RoboDK station: KUKA.rdk

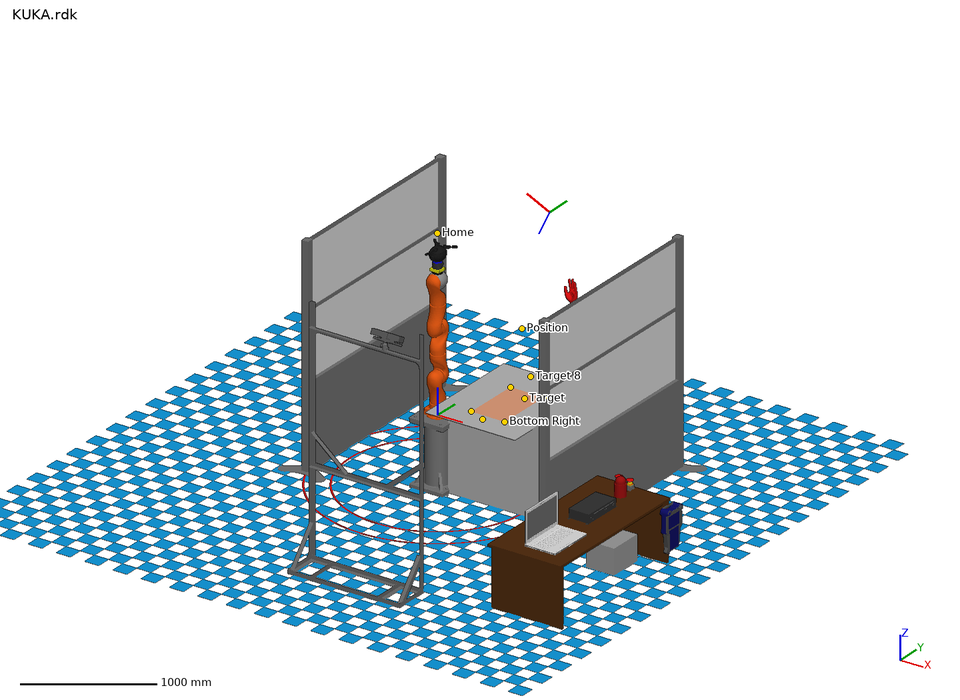
[picture v0: the station drawn from its stored meshes, robots at their saved joint values, targets as dots, program paths as lines]
Station robotSim. Poses are relative to the parent item; angles as X-Y-Z fixed-axis rotations.
Station parameters (name, value as stored): IO_5, 1
  - frame KUKA-LWR-IV-PLUS Base at (0, 0, 570) mm
    - robot KUKA: 7 axes
        modified DH rows (alpha deg, a mm, theta deg, d mm): 0, 0, 0, 310.5; -90, 0, -90, 0; 90, 0, 0, 400; -90, 0, 0, 0; 90, 0, 0, 390; -90, 0, 0, 0; 90, 0, 0, 78
        joint limits [-170, -30, -170, -120, -170, -120, -170] to [170, 210, 170, 120, 170, 120, 170]; home [0, 90, 0, 0, 0, 0, 0]; saved at [0, 90, 0, 0, 0, 0, 0]
      - tool Gripper, TCP at (0, 0, 300) mm, size 214.4 x 261.8 x 207.2 mm, geometry from FULL_GRIPPER_ATI.stl
    - target Target (Cartesian target) at (600, 250, 200) mm, rotated rx -90 ry 0 rz 0 deg; joints [-12.043, 152.871, 0, -75.808, -99.102, -97.918, -49.31] of KUKA
    - target Bottom Right (Cartesian target) at (705, -150, 200) mm, rotated rx 180 ry 0 rz -135 deg; joints [-12.011, 146.511, 0, -26.598, 0, 96.891, -57.011] of KUKA
    - target Bottom Left (Cartesian target) at (405, -150, 200) mm, rotated rx 180 ry 0 rz 135 deg; joints [-20.323, 99.106, 0, -99.97, 0, 70.924, 24.677] of KUKA
    - target Top Left (Cartesian target) at (405, 350, 200) mm, rotated rx 180 ry 0 rz 45 deg; joints [-139.167, 66.69, 0, 81.525, 0, -75.165, -4.167] of KUKA
    - target Top Right (Cartesian target) at (705, 350, 200) mm, rotated rx 180 ry 0 rz -45 deg; joints [-134.648, 29.334, 0, 17.033, 0, -102.301, 90.352] of KUKA
    - target Position (Cartesian target) at (570, 260, 760) mm, rotated rx -90 ry 0 rz 0 deg; joints [-7.407, 162.566, 0, 37.615, 96.082, 94.235, -124.726] of KUKA
    - target Target 8 (Cartesian target) at (585, 350, 335) mm, rotated rx 180 ry 0 rz 45 deg; joints [-150.368, 51.861, 0, 38.836, 0, -103.025, -15.368] of KUKA
    - frame Light Source at (1000, 0, 1930) mm, rotated rx 180 ry -25 rz 180 deg
    - target Test (joint target) at (545, -205, 200) mm, rotated rx 165 ry 0 rz 45 deg; joints [-15.931, 108.28, 0, -90.444, -8.492, 58.378, 122.709] of KUKA
    - target Home (Cartesian target) at (0, 0, 1478.5) mm; joints [0, 90, 0, 0, 0, 0, 0] of KUKA
    - object Sheet at (555, 100, 200) mm, rotated rx 0 ry 0 rz 90 deg, size 500 x 300 x 0.1 mm, geometry from Sheet.stl
  - object Base at (0, 0, 0) mm, size 305 x 305 x 604 mm, geometry from Base.stl
  - object Plane at (0, 0, 0) mm, size 5042.2 x 5042.2 x 2.5 mm, geometry from plane_1m_grid.sld
  - object ATI_FT_Controller at (1800, -600, 520) mm, rotated rx 0 ry 0 rz -90 deg, size 383.6 x 183 x 76 mm, geometry from ATI_FT_Controller.stl
  - object Kinect at (620, -1500, 1985) mm, rotated rx -119.64 ry 0 rz 0 deg, size 250 x 70 x 76 mm, geometry from Kinect.stl
  - object Camera_Base at (620, -1560, 1962) mm, rotated rx 0 ry 0 rz -90 deg, size 300 x 1000 x 2100 mm, geometry from Camera_Base.stl
  - object Wall1 at (1270, 400, 0) mm, rotated rx 0 ry 0 rz 90 deg, size 1940 x 400 x 1880 mm, geometry from Wall_stripped.stl
  - object Glass1.1 at (1270, 400, 1008) mm, rotated rx 0 ry 0 rz 90 deg, size 1640 x 10 x 555 mm, geometry from Glass1.stl
  - object Glass1.2 at (1270, 400, 1582) mm, rotated rx 0 ry 0 rz 90 deg, size 1640 x 10 x 535 mm, geometry from Glass2.stl
  - object Wall2 at (-920, 500, 0) mm, rotated rx 0 ry 0 rz 90 deg, size 1940 x 400 x 1880 mm, geometry from Wall_stripped.stl
  - object Glass2.1 at (-920, 500, 1008) mm, rotated rx 0 ry 0 rz 90 deg, size 1640 x 10 x 555 mm, geometry from Glass1.stl
  - object Glass2.2 at (-920, 500, 1582) mm, rotated rx 0 ry 0 rz 90 deg, size 1640 x 10 x 535 mm, geometry from Glass2.stl
  - object Table at (535, 150, 0) mm, size 800 x 1000 x 770 mm, geometry from Table.stl
  - object Desk at (1800, -770, 520) mm, rotated rx 0 ry 0 rz -90 deg, size 1400 x 650 x 520 mm, geometry from Desk.stl
  - object Laptop at (2000, -950, 520) mm, rotated rx 90 ry 0 rz 90 deg, size 411 x 298 x 272.1 mm, geometry from Laptop.stl
  - object Safety Light at (1800, -250, 470) mm, rotated rx 90 ry 0 rz 0 deg, size 94.9 x 207.5 x 95 mm, geometry from Safety Light.STL
  - object Teach Pendant at (2150, -100, 300) mm, rotated rx 90 ry 0 rz 90 deg, size 203.1 x 365.4 x 82.6 mm, geometry from Teach Pendant.stl
  - object KUKA_Computer at (1800, -350, 0) mm, rotated rx 0 ry 0 rz 90 deg, size 300 x 250 x 220 mm, geometry from KUKA_Computer.stl
  - object Hand at (500, 1000, 1400) mm, rotated rx 0 ry 0 rz -90 deg, size 224.5 x 118 x 62.6 mm, geometry from Hand.stl
  - object Kuka_workspace at (0, 0, 1.5) mm, size 1580 x 1580 x 0.1 mm, geometry from kuka_workspace.stl
  - object Gripper_workspace at (0, 0, 1.5) mm, size 1980 x 1979.6 x 0.1 mm, geometry from gripper_workspace.stl
  - object Emergency_button_1 at (1775, -130, 477) mm, rotated rx 90 ry 0 rz 0 deg, size 55.1 x 89.2 x 55.1 mm, geometry from emergency_button.stl
  - object Emergency_button_2 at (1675, -130, 477) mm, rotated rx 90 ry 0 rz 0 deg, size 55.1 x 89.2 x 55.1 mm, geometry from Emergency_button.stl
  - object CloudSkeletonParticles at (0, 1500, 1000) mm, size 29.8 x 30 x 29.8 mm, geometry from particle.stl
    - object FACE at (0, 0, 0) mm, size 29.8 x 30 x 29.8 mm, geometry from particle.stl
      - object HEAD at (100, 0, 0) mm, size 29.8 x 30 x 29.8 mm, geometry from particle.stl
      - object NECK at (96.86, 0, 24.87) mm, size 29.8 x 30 x 29.8 mm, geometry from particle.stl
    - object SPINE at (0, 0, 0) mm, size 29.8 x 30 x 29.8 mm, geometry from particle.stl
      - object SPINE_SHOULDER at (87.63, 0, 48.18) mm, size 29.8 x 30 x 29.8 mm, geometry from particle.stl
      - object SPINE_MID at (72.9, 0, 68.45) mm, size 29.8 x 30 x 29.8 mm, geometry from particle.stl
      - object SPINE_BASE at (53.58, 0, 84.43) mm, size 29.8 x 30 x 29.8 mm, geometry from particle.stl
    - object RIGHT_ARM at (0, 0, 0) mm, size 29.8 x 30 x 29.8 mm, geometry from particle.stl
      - object SHOULDER_RIGHT at (30.9, 0, 95.11) mm, size 29.8 x 30 x 29.8 mm, geometry from particle.stl
      - object ELBOW_RIGHT at (6.28, 0, 99.8) mm, size 29.8 x 30 x 29.8 mm, geometry from particle.stl
      - object WRIST_RIGHT at (-18.74, 0, 98.23) mm, size 29.8 x 30 x 29.8 mm, geometry from particle.stl
      - object HAND_RIGHT at (-42.58, 0, 90.48) mm, size 29.8 x 30 x 29.8 mm, geometry from particle.stl
      - object THUMB_RIGHT at (-63.74, 0, 77.05) mm, size 29.8 x 30 x 29.8 mm, geometry from particle.stl
      - object HAND_TIP_RIGHT at (-80.9, 0, 58.78) mm, size 29.8 x 30 x 29.8 mm, geometry from particle.stl
    - object LEFT_ARM at (0, 0, 0) mm, size 29.8 x 30 x 29.8 mm, geometry from particle.stl
      - object SHOULDER_LEFT at (-92.98, 0, 36.81) mm, size 29.8 x 30 x 29.8 mm, geometry from particle.stl
      - object ELBOW_LEFT at (-99.21, 0, 12.53) mm, size 29.8 x 30 x 29.8 mm, geometry from particle.stl
      - object WRIST_LEFT at (-99.21, 0, -12.53) mm, size 29.8 x 30 x 29.8 mm, geometry from particle.stl
      - object HAND_LEFT at (-92.98, 0, -36.81) mm, size 29.8 x 30 x 29.8 mm, geometry from particle.stl
      - object THUMB_LEFT at (-80.9, 0, -58.78) mm, size 29.8 x 30 x 29.8 mm, geometry from particle.stl
      - object HAND_TIP_LEFT at (-63.74, 0, -77.05) mm, size 29.8 x 30 x 29.8 mm, geometry from particle.stl
    - object LEG_RIGHT at (0, 0, 0) mm, size 29.8 x 30 x 29.8 mm, geometry from particle.stl
      - object HIP_RIGHT at (-42.58, 0, -90.48) mm, size 29.8 x 30 x 29.8 mm, geometry from particle.stl
      - object KNEE_RIGHT at (-18.74, 0, -98.23) mm, size 29.8 x 30 x 29.8 mm, geometry from particle.stl
      - object ANKLE_RIGHT at (6.28, 0, -99.8) mm, size 29.8 x 30 x 29.8 mm, geometry from particle.stl
      - object FOOT_RIGHT at (30.9, 0, -95.11) mm, size 29.8 x 30 x 29.8 mm, geometry from particle.stl
    - object LEG_LEFT at (0, 0, 0) mm, size 29.8 x 30 x 29.8 mm, geometry from particle.stl
      - object HIP_LEFT at (53.58, 0, -84.43) mm, size 29.8 x 30 x 29.8 mm, geometry from particle.stl
      - object KNEE_LEFT at (72.9, 0, -68.45) mm, size 29.8 x 30 x 29.8 mm, geometry from particle.stl
      - object ANKLE_LEFT at (87.63, 0, -48.18) mm, size 29.8 x 30 x 29.8 mm, geometry from particle.stl
      - object FOOT_LEFT at (96.86, 0, -24.87) mm, size 29.8 x 30 x 29.8 mm, geometry from particle.stl
  - Python program testing (listed below)
  - Python program Prog2 (listed below)
  - Python program Prog3 (listed below)
  - Python program Prog4 (listed below)
  - Python program Prog8 (listed below)
  - Python program goHome (listed below)
  - Python program Reset Cloud Skeleton (listed below)
  - Python program Reset (listed below)
  - Python program testCamera (listed below)
  - Python program CloudSkeletonReset (listed below)
  - Python program TestConnection (listed below)
  - Python program testRobotItem (listed below)
  - Python program testJoints (listed below)
  - Python program testRot (listed below)
  - Python program testFabric (listed below)
  - Python program quasi (listed below)
  - Python program transient (listed below)
  - Python program testJointLimits (listed below)

--- Python program testing ---
from robolink.robolink import Robolink
from robodk.robodk import Pose_2_KUKA, KUKA_2_Pose, rotz, tr

RDK = Robolink()

# Turn off automatic rendering (faster simulation)
RDK.Render(False)

robot = RDK.Item("KUKA")
pose = RDK.Item('Target')
tl = RDK.Item('Top Left')
target = Pose_2_KUKA(tl.Pose())
tl.setPose(KUKA_2_Pose((target[0], target[1], target[2] + 10, target[3], target[4], target[5])))
# robot.MoveJ(pose)
RDK.Render(True)

--- Python program Prog2 ---
# Type help("robolink") or help("robodk") for more information
# Press F5 to run the script
# Documentation: https://robodk.com/doc/en/RoboDK-API.html
# Reference:     https://robodk.com/doc/en/PythonAPI/index.html
# Note: It is not required to keep a copy of this file, your python script is saved with the station
from robolink import *    # RoboDK API
from robodk import *      # Robot toolbox
RDK = Robolink()

robot = RDK.Item("KUKA")
pose = RDK.Item("Target")
pose.setPose(KUKA_2_Pose(list((100, 200, 300,  0, 0, 0))))

issues = robot.MoveJ_Test(robot.Joints(), pose.Joints())
can_move_joints = (issues == 0)
if can_move_joints:
    # Move Robot
    robot.MoveJ(pose)
    # Update robot state
    robot_state = 'MOVING'

--- Python program Prog3 ---
# Type help("robolink") or help("robodk") for more information
# Press F5 to run the script
# Documentation: https://robodk.com/doc/en/RoboDK-API.html
# Reference:     https://robodk.com/doc/en/PythonAPI/index.html
# Note: It is not required to keep a copy of this file, your python script is saved with the station
from robolink import *    # RoboDK API
from robodk import *      # Robot toolbox
import math
RDK = Robolink()

light = RDK.Item('Light Source')
light.setPoseAbs(KUKA_2_Pose(list((1000, 0, 2500, 0, 205, 0))))

#RDK.setFlagsRoboDK(flags=[FLAG_ROBODK_TREE_ACTIVE, FLAG_ROBODK_3DVIEW_ACTIVE, FLAG_ROBODK_LEFT_CLICK, FLAG_ROBODK_RIGHT_CLICK, FLAG_ROBODK_DOUBLE_CLICK ])

--- Python program Prog4 ---
# Type help("robolink") or help("robodk") for more information
# Press F5 to run the script
# Documentation: https://robodk.com/doc/en/RoboDK-API.html
# Reference:     https://robodk.com/doc/en/PythonAPI/index.html
# Note: It is not required to keep a copy of this file, your python script is saved with the station
from robolink import *    # RoboDK API
from robodk import *      # Robot toolbox
RDK = Robolink()
"""
RDK.Command('CollisionMethod', value='CUDA')
RDK.Command('DisplayCurves', value='0')
RDK.Command('SetSize3D', value='650x610')
RDK.Command('Trace', value='On')
"""
kinect = RDK.Item('Kinect')  # Get Kinect
# Define Camera
# Close all cameras just in case
RDK.Cam2D_Close()
# Pick which items will act as the camera
# camref = RDK.ItemUserPick('Select the camera')
# Use the GLSL files for more realistic camera view from inside the RoboDK software
file_shader_fragment = 'D:/Downloads/Kinect python/RoboDK/KUKA/Camera-Shaders/shader_fragment.glsl'
file_shader_vertex = 'D:/Downloads/Kinect python/RoboDK/KUKA/Camera-Shaders/shader_vertex.glsl'
# Add Camera
"""
# -------------Set parameters in mm and degrees-------------------------
#  FOV: Field of view in degrees (atan(0.5*height/distance) of the sensor
#  FOCAL_LENGTH: focal length in mm
#  FAR_LENGTH: maximum working distance (in mm)
#  SIZE: size of the window in pixels (fixed) (width x height)
#  SNAPSHOT: size of the snapshot image in pixels (width x height)
#  BG_COLOR: background color (rgb color or named color: AARRGGBB)
#  LIGHT_AMBIENT: ambient color (rgb color or named color: AARRGGBB)
#  LIGHT_SPECULAR: specular color (rgb color or named color: AARRGGBB)
#  LIGHT_DIFFUSE: diffuse color (rgb color or named color: AARRGGBB)
#  DEPTH: Add this flag to create a 32 bit depth map (white=close, black=far)
#  NO_TASKBAR: Don't add the window to the task bar
#  MINIMIZED: Show the window minimized
#  ALWAYS_VISIBLE: Keep the window on top of all other windows
#  SHADER_VERTEX: File to a vertex shader (GLSL file)
#  SHADER_FRAGMENT: File to a fragment shader (GLSL file)
"""
# cam_id = RDK.Cam2D_Add(kinect, 'FOCAL_LENGTH=' + str(focal_length) + ' FOV=' + str(field_of_view) + ' FAR_LENGTH=4500 SIZE=548x308 BG_COLOR=black LIGHT_AMBIENT=red LIGHT_DIFFUSE=black LIGHT_SPECULAR=white ALWAYS_VISIBLE')
# RDK.Cam2D_Add(kinect, 'FOCAL_LENGTH=' + str(focal_length) + ' FOV=' + str(field_of_view) + ' FAR_LENGTH=4500 SIZE=548x308 BG_COLOR=black LIGHT_AMBIENT=red LIGHT_DIFFUSE=black LIGHT_SPECULAR=white TASKBAR ALWAYS_VISIBLE')
RDK.Cam2D_Add(kinect, 'FOCAL_LENGTH=1000 FOV=60 FAR_LENGTH=4500 SIZE=548x308 BG_COLOR=black SHADER_FRAGMENT=' + file_shader_fragment + ' SHADER_VERTEX=' + file_shader_vertex)
# Special command to retrieve the window ID:

--- Python program Prog8 ---
from robolink import *    # RoboDK API
from robodk import *      # Robot toolbox
RDK = Robolink()
RDK.setRunMode(6)
robot = RDK.Item('KUKA')
home = RDK.Item("Home")
bl = RDK.Item('Bottom Left')
j = tr(bl.Joints())
#print(j[0,0], j[0,1], j[0, 2], j[0,3], j[0,4], j[0,5], j[0,6])
robot.MoveJ(home)

robot.MoveJ([j[0, 0], j[0, 1], j[0, 3], j[0, 4], j[0, 5], j[0, 6], j[0, 2]])

#robot.MoveJ(home)

--- Python program goHome ---
# Type help("robolink") or help("robodk") for more information
# Press F5 to run the script
# Documentation: https://robodk.com/doc/en/RoboDK-API.html
# Reference:     https://robodk.com/doc/en/PythonAPI/index.html
# Note: It is not required to keep a copy of this file, your python script is saved with the station
from robolink import *    # RoboDK API
from robodk import *      # Robot toolbox
RDK = Robolink()
RDK.setRunMode(6)
robot = RDK.Item('KUKA')
robot.MoveJ([0, 90, 0, 0, 0, 0, 0])

--- Python program Reset Cloud Skeleton ---
from robolink import *    # RoboDK API
from robodk import *      # Robot toolbox
RDK = Robolink()

--- Python program Reset ---
# Type help("robolink") or help("robodk") for more information
# Press F5 to run the script
# Documentation: https://robodk.com/doc/en/RoboDK-API.html
# Reference:     https://robodk.com/doc/en/PythonAPI/index.html
# Note: It is not required to keep a copy of this file, your python script is saved with the station
from robolink import *    # RoboDK API
from robodk import *      # Robot toolbox
RDK = Robolink()

sheet = RDK.Item('Sheet')  # Sheet item
pose = RDK.Item('Target')  # Target
br = RDK.Item('Bottom Right')  # Bottom Right Corner of Fabric
bl = RDK.Item('Bottom Left')  # Bottom Left Corner of Fabric
tl = RDK.Item('Top Left')  # Top Left Corner of Fabric
tr = RDK.Item('Top Right')  # Top Right Corner of Fabric
hand = RDK.Item('Hand')  # Get hand model
robot = RDK.Item('KUKA')  # Get Robot Model
RDK.RunCode('CloudSkeletonReset', True)  # Reset CloudSkeleton
# Reset Robot
robot.setJoints([0, 90, 0, 0, 0, 0])

# Reset Sheet
sheet.Delete()
sheet = RDK.AddFile(r'D:\Downloads\KinectPython\Models\Sheet.stl')
sheet.setPoseAbs(KUKA_2_Pose(list((555, 100, 770, 90, 0, 0))))
sheet.setColor([255/255, 170/255, 127/255, 1])


br.setPoseAbs(KUKA_2_Pose(list((705, -150, 770, 45, -180, 0))))
bl.setPoseAbs(KUKA_2_Pose(list((405, -150, 770, -45, 180, 0))))
tl.setPoseAbs(KUKA_2_Pose(list((405, 350, 770, 45, 0, 180))))
tr.setPoseAbs(KUKA_2_Pose(list((705, 350, 770, -45, 0, 180))))

# Reset Hand
hand.setPoseAbs(KUKA_2_Pose(list((500, 1000, 1400, -90, 0, 0))))

# Reset Target
pose.setPoseAbs(KUKA_2_Pose(list((600, 250, 770, 0, 0, -90))))

--- Python program testCamera ---
from robolink import *    # RoboDK API
from robodk import *      # Robot toolbox
RDK = Robolink()

kinect = RDK.Item('Kinect')  # Get Kinect
light = RDK.Item('Light Source')  # Get Light Source

# Use the GLSL files for more realistic camera view from inside the RoboDK software
file_shader_fragment = 'D:/Downloads/Kinect python/RoboDK/KUKA/Camera-Shaders/shader_fragment.glsl'
file_shader_vertex = 'D:/Downloads/Kinect python/RoboDK/KUKA/Camera-Shaders/shader_vertex.glsl'
RDK.Cam2D_Add(kinect, 'FOCAL_LENGTH=1064.3187 FOV=38.011 FAR_LENGTH=4500 SIZE=512x424 BG_COLOR=default SHADER_FRAGMENT=' + file_shader_fragment + ' SHADER_VERTEX=' + file_shader_vertex)

--- Python program CloudSkeletonReset ---
from robolink import *    # RoboDK API
from robodk import *      # Robot toolbox
import math
RDK = Robolink()
OFFSET_RGB = 95  # mm
CLOUD_RESET_RADIUS = 100  # mm
PARTICLE_RADIUS = 30  # mm

kinect_model = RDK.Item('Kinect')


# Class to represent the Operator
class CloudSkeleton(object):

    def __init__(self):
        # Initialize the operator Skeleton

        # HEAD
        self.HEAD = RDK.Item('HEAD')
        self.NECK = RDK.Item('NECK')

        # SPINE
        self.SPINE_SHOULDER = RDK.Item('SPINE_SHOULDER')
        self.SPINE_MID = RDK.Item('SPINE_MID')
        self.SPINE_BASE = RDK.Item('SPINE_BASE')

        # RIGHT ARM
        self.SHOULDER_RIGHT = RDK.Item('SHOULDER_RIGHT')
        self.ELBOW_RIGHT = RDK.Item('ELBOW_RIGHT')
        self.WRIST_RIGHT = RDK.Item('WRIST_RIGHT')
        self.HAND_RIGHT = RDK.Item('HAND_RIGHT')
        self.THUMB_RIGHT = RDK.Item('THUMB_RIGHT')
        self.HAND_TIP_RIGHT = RDK.Item('HAND_TIP_RIGHT')

        # LEFT ARM
        self.SHOULDER_LEFT = RDK.Item('SHOULDER_LEFT')
        self.ELBOW_LEFT = RDK.Item('ELBOW_LEFT')
        self.WRIST_LEFT = RDK.Item('WRIST_LEFT')
        self.HAND_LEFT = RDK.Item('HAND_LEFT')
        self.THUMB_LEFT = RDK.Item('THUMB_LEFT')
        self.HAND_TIP_LEFT = RDK.Item('HAND_TIP_LEFT')

        # LEG RIGHT
        self.HIP_RIGHT = RDK.Item('HIP_RIGHT')
        self.KNEE_RIGHT = RDK.Item('KNEE_RIGHT')
        self.ANKLE_RIGHT = RDK.Item('ANKLE_RIGHT')
        self.FOOT_RIGHT = RDK.Item('FOOT_RIGHT')

        # LEG LEFT
        self.HIP_LEFT = RDK.Item('HIP_LEFT')
        self.KNEE_LEFT = RDK.Item('KNEE_LEFT')
        self.ANKLE_LEFT = RDK.Item('ANKLE_LEFT')
        self.FOOT_LEFT = RDK.Item('FOOT_LEFT')

        # Full Body and All Joints
        self.Body = RDK.Item('CloudSkeletonParticles')
        self.Joints = RDK.Item('CloudSkeletonParticles').Childs()

        # Reset the position of all the particles for easier translation
        self.Body.setPoseAbs(KUKA_2_Pose(list((0, 1500, 1000, 0, 0, 0))))

        # Set the Skeleton's Color
        # -------------- Color = [r, g, b, a] (from 0 to 1 scale) (a = opacity, 0=transparent, 1=solid)
        for joints in self.Joints:
            for particle in joints.Childs():
                particle.setColor([255/255, 0/255, 255/255, 1])

    def Circle(self):
        RDK.Render(False)
        # Find Number of particles
        n_particles = 0
        for joints in self.Joints:
            for particle in joints.Childs():
                n_particles += 1

        # Reset the Position of the Cloud Skeleton
        counter = 0
        for joints in self.Joints:
            for particle in joints.Childs():
                particle.setPose(KUKA_2_Pose(list((CLOUD_RESET_RADIUS*math.cos(counter*2*math.pi/n_particles), 0, CLOUD_RESET_RADIUS*math.sin(counter*2*math.pi/n_particles), 0, 0, 0))))
                counter += 1
        RDK.Render(True)

    def Torus(self):
        RDK.Render(False)
        # Find Number of particles
        n_particles = 0
        for joints in self.Joints:
            for particle in joints.Childs():
                n_particles += 1

        # Reset the Position of the Cloud Skeleton
        counter = 0
        for joints in self.Joints:
            for particle in joints.Childs():
                particle.setPose(KUKA_2_Pose(list((PARTICLE_RADIUS*math.cos(counter*2*math.pi/n_particles), 0, PARTICLE_RADIUS*math.sin(counter*2*math.pi/n_particles), 0, 0, 0))))
                counter += 1
        RDK.Render(True)

    def Visible(self):
        RDK.Render(False)  # Faster Computations
        # Make CloudSkeleton Visible
        for joints in self.Joints:
            for particle in joints.Childs():
                particle.setVisible(1)
        RDK.Render(True)

    def Invisible(self):
        RDK.Render(False)  # Faster Computations
        # Make CloudSkeleton Invisible
        for joints in self.Joints:
            for particle in joints.Childs():
                particle.setVisible(0)
        RDK.Render(True)

    def Update(self, joints, kinect_model):
        RDK.Render(False)  # Faster Computations

        # Update CloudSkeletonParticles with real world coordinates of joints

        # HEAD
        HEAD_POSE = Pose_2_KUKA(kinect_model.Pose()*transl(-joints[PyKinectV2.JointType_Head].Position.x*1000, -joints[PyKinectV2.JointType_Head].Position.y*1000, joints[PyKinectV2.JointType_Head].Position.z*1000))
        NECK_POSE = Pose_2_KUKA(kinect_model.Pose()*transl(-joints[PyKinectV2.JointType_Neck].Position.x*1000, -joints[PyKinectV2.JointType_Neck].Position.y*1000, joints[PyKinectV2.JointType_Neck].Position.z*1000))
        self.HEAD.setPoseAbs(KUKA_2_Pose(list((HEAD_POSE[0] + OFFSET_RGB, HEAD_POSE[1], HEAD_POSE[2], 0, 0, 0))))
        self.NECK.setPoseAbs(KUKA_2_Pose(list((NECK_POSE[0] + OFFSET_RGB, NECK_POSE[1], NECK_POSE[2], 0, 0, 0))))

        # SPINE
        SPINE_SHOULDER_POSE = Pose_2_KUKA(kinect_model.Pose()*transl(-joints[PyKinectV2.JointType_SpineShoulder].Position.x*1000, -joints[PyKinectV2.JointType_SpineShoulder].Position.y*1000, joints[PyKinectV2.JointType_SpineShoulder].Position.z*1000))
        SPINE_MID_POSE = Pose_2_KUKA(kinect_model.Pose()*transl(-joints[PyKinectV2.JointType_SpineMid].Position.x*1000, -joints[PyKinectV2.JointType_SpineMid].Position.y*1000, joints[PyKinectV2.JointType_SpineMid].Position.z*1000))
        SPINE_BASE_POSE = Pose_2_KUKA(kinect_model.Pose()*transl(-joints[PyKinectV2.JointType_SpineBase].Position.x*1000, -joints[PyKinectV2.JointType_SpineBase].Position.y*1000, joints[PyKinectV2.JointType_SpineBase].Position.z*1000))
        self.SPINE_SHOULDER.setPoseAbs(KUKA_2_Pose(list((SPINE_SHOULDER_POSE[0] + OFFSET_RGB, SPINE_SHOULDER_POSE[1], SPINE_SHOULDER_POSE[2], 0, 0, 0))))
        self.SPINE_MID.setPoseAbs(KUKA_2_Pose(list((SPINE_MID_POSE[0] + OFFSET_RGB, SPINE_MID_POSE[1], SPINE_MID_POSE[2], 0, 0, 0))))
        self.SPINE_BASE.setPoseAbs(KUKA_2_Pose(list((SPINE_BASE_POSE[0] + OFFSET_RGB, SPINE_BASE_POSE[1], SPINE_BASE_POSE[2], 0, 0, 0))))

        # RIGHT ARM
        SHOULDER_RIGHT_POSE = Pose_2_KUKA(kinect_model.Pose()*transl(-joints[PyKinectV2.JointType_ShoulderRight].Position.x*1000, -joints[PyKinectV2.JointType_ShoulderRight].Position.y*1000, joints[PyKinectV2.JointType_ShoulderRight].Position.z*1000))
        ELBOW_RIGHT_POSE = Pose_2_KUKA(kinect_model.Pose()*transl(-joints[PyKinectV2.JointType_ElbowRight].Position.x*1000, -joints[PyKinectV2.JointType_ElbowRight].Position.y*1000, joints[PyKinectV2.JointType_ElbowRight].Position.z*1000))
        WRIST_RIGHT_POSE = Pose_2_KUKA(kinect_model.Pose()*transl(-joints[PyKinectV2.JointType_WristRight].Position.x*1000, -joints[PyKinectV2.JointType_WristRight].Position.y*1000, joints[PyKinectV2.JointType_WristRight].Position.z*1000))
        HAND_RIGHT_POSE = Pose_2_KUKA(kinect_model.Pose()*transl(-joints[PyKinectV2.JointType_HandRight].Position.x*1000, -joints[PyKinectV2.JointType_HandRight].Position.y*1000, joints[PyKinectV2.JointType_HandRight].Position.z*1000))
        THUMB_RIGHT_POSE = Pose_2_KUKA(kinect_model.Pose()*transl(-joints[PyKinectV2.JointType_ThumbRight].Position.x*1000, -joints[PyKinectV2.JointType_ThumbRight].Position.y*1000, joints[PyKinectV2.JointType_ThumbRight].Position.z*1000))
        HAND_TIP_RIGHT_POSE = Pose_2_KUKA(kinect_model.Pose()*transl(-joints[PyKinectV2.JointType_HandTipRight].Position.x*1000, -joints[PyKinectV2.JointType_HandTipRight].Position.y*1000, joints[PyKinectV2.JointType_HandTipRight].Position.z*1000))
        self.SHOULDER_RIGHT.setPoseAbs(KUKA_2_Pose(list((SHOULDER_RIGHT_POSE[0] + OFFSET_RGB, SHOULDER_RIGHT_POSE[1], SHOULDER_RIGHT_POSE[2], 0, 0, 0))))
        self.ELBOW_RIGHT.setPoseAbs(KUKA_2_Pose(list((ELBOW_RIGHT_POSE[0] + OFFSET_RGB, ELBOW_RIGHT_POSE[1], ELBOW_RIGHT_POSE[2], 0, 0, 0))))
        self.WRIST_RIGHT.setPoseAbs(KUKA_2_Pose(list((WRIST_RIGHT_POSE[0] + OFFSET_RGB, WRIST_RIGHT_POSE[1], WRIST_RIGHT_POSE[2], 0, 0, 0))))
        self.HAND_RIGHT.setPoseAbs(KUKA_2_Pose(list((HAND_RIGHT_POSE[0] + OFFSET_RGB, HAND_RIGHT_POSE[1], HAND_RIGHT_POSE[2], 0, 0, 0))))
        self.THUMB_RIGHT.setPoseAbs(KUKA_2_Pose(list((THUMB_RIGHT_POSE[0] + OFFSET_RGB, THUMB_RIGHT_POSE[1], THUMB_RIGHT_POSE[2], 0, 0, 0))))
        self.HAND_TIP_RIGHT.setPoseAbs(KUKA_2_Pose(list((HAND_TIP_RIGHT_POSE[0] + OFFSET_RGB, HAND_TIP_RIGHT_POSE[1], HAND_TIP_RIGHT_POSE[2], 0, 0, 0))))

        # LEFT ARM
        SHOULDER_LEFT_POSE = Pose_2_KUKA(kinect_model.Pose()*transl(-joints[PyKinectV2.JointType_ShoulderLeft].Position.x*1000, -joints[PyKinectV2.JointType_ShoulderLeft].Position.y*1000, joints[PyKinectV2.JointType_ShoulderLeft].Position.z*1000))
        ELBOW_LEFT_POSE = Pose_2_KUKA(kinect_model.Pose()*transl(-joints[PyKinectV2.JointType_ElbowLeft].Position.x*1000, -joints[PyKinectV2.JointType_ElbowLeft].Position.y*1000, joints[PyKinectV2.JointType_ElbowLeft].Position.z*1000))
        WRIST_LEFT_POSE = Pose_2_KUKA(kinect_model.Pose()*transl(-joints[PyKinectV2.JointType_WristLeft].Position.x*1000, -joints[PyKinectV2.JointType_WristLeft].Position.y*1000, joints[PyKinectV2.JointType_WristLeft].Position.z*1000))
        HAND_LEFT_POSE = Pose_2_KUKA(kinect_model.Pose()*transl(-joints[PyKinectV2.JointType_HandLeft].Position.x*1000, -joints[PyKinectV2.JointType_HandLeft].Position.y*1000, joints[PyKinectV2.JointType_HandLeft].Position.z*1000))
        THUMB_LEFT_POSE = Pose_2_KUKA(kinect_model.Pose()*transl(-joints[PyKinectV2.JointType_ThumbLeft].Position.x*1000, -joints[PyKinectV2.JointType_ThumbLeft].Position.y*1000, joints[PyKinectV2.JointType_ThumbLeft].Position.z*1000))
        HAND_TIP_LEFT_POSE = Pose_2_KUKA(kinect_model.Pose()*transl(-joints[PyKinectV2.JointType_HandTipLeft].Position.x*1000, -joints[PyKinectV2.JointType_HandTipLeft].Position.y*1000, joints[PyKinectV2.JointType_HandTipLeft].Position.z*1000))
        self.SHOULDER_LEFT.setPoseAbs(KUKA_2_Pose(list((SHOULDER_LEFT_POSE[0] + OFFSET_RGB, SHOULDER_LEFT_POSE[1], SHOULDER_LEFT_POSE[2], 0, 0, 0))))
        self.ELBOW_LEFT.setPoseAbs(KUKA_2_Pose(list((ELBOW_LEFT_POSE[0] + OFFSET_RGB, ELBOW_LEFT_POSE[1], ELBOW_LEFT_POSE[2], 0, 0, 0))))
        self.WRIST_LEFT.setPoseAbs(KUKA_2_Pose(list((WRIST_LEFT_POSE[0] + OFFSET_RGB, WRIST_LEFT_POSE[1], WRIST_LEFT_POSE[2], 0, 0, 0))))
        self.HAND_LEFT.setPoseAbs(KUKA_2_Pose(list((HAND_LEFT_POSE[0] + OFFSET_RGB, HAND_LEFT_POSE[1], HAND_LEFT_POSE[2], 0, 0, 0))))
        self.THUMB_LEFT.setPoseAbs(KUKA_2_Pose(list((THUMB_LEFT_POSE[0] + OFFSET_RGB, THUMB_LEFT_POSE[1], THUMB_LEFT_POSE[2], 0, 0, 0))))
        self.HAND_TIP_LEFT.setPoseAbs(KUKA_2_Pose(list((HAND_TIP_LEFT_POSE[0] + OFFSET_RGB, HAND_TIP_LEFT_POSE[1], HAND_TIP_LEFT_POSE[2], 0, 0, 0))))

        # LEG RIGHT
        HIP_RIGHT_POSE = Pose_2_KUKA(kinect_model.Pose()*transl(-joints[PyKinectV2.JointType_HipRight].Position.x*1000, -joints[PyKinectV2.JointType_HipRight].Position.y*1000, joints[PyKinectV2.JointType_HipRight].Position.z*1000))
        KNEE_RIGHT_POSE = Pose_2_KUKA(kinect_model.Pose()*transl(-joints[PyKinectV2.JointType_KneeRight].Position.x*1000, -joints[PyKinectV2.JointType_KneeRight].Position.y*1000, joints[PyKinectV2.JointType_KneeRight].Position.z*1000))
        ANKLE_RIGHT_POSE = Pose_2_KUKA(kinect_model.Pose()*transl(-joints[PyKinectV2.JointType_AnkleRight].Position.x*1000, -joints[PyKinectV2.JointType_AnkleRight].Position.y*1000, joints[PyKinectV2.JointType_AnkleRight].Position.z*1000))
        FOOT_RIGHT_POSE = Pose_2_KUKA(kinect_model.Pose()*transl(-joints[PyKinectV2.JointType_FootRight].Position.x*1000, -joints[PyKinectV2.JointType_FootRight].Position.y*1000, joints[PyKinectV2.JointType_FootRight].Position.z*1000))
        self.HIP_RIGHT.setPoseAbs(KUKA_2_Pose(list((HIP_RIGHT_POSE[0] + OFFSET_RGB, HIP_RIGHT_POSE[1], HIP_RIGHT_POSE[2], 0, 0, 0))))
        self.KNEE_RIGHT.setPoseAbs(KUKA_2_Pose(list((KNEE_RIGHT_POSE[0] + OFFSET_RGB, KNEE_RIGHT_POSE[1], KNEE_RIGHT_POSE[2], 0, 0, 0))))
        self.ANKLE_RIGHT.setPoseAbs(KUKA_2_Pose(list((ANKLE_RIGHT_POSE[0] + OFFSET_RGB, ANKLE_RIGHT_POSE[1], ANKLE_RIGHT_POSE[2], 0, 0, 0))))
        self.FOOT_RIGHT.setPoseAbs(KUKA_2_Pose(list((FOOT_RIGHT_POSE[0] + OFFSET_RGB, FOOT_RIGHT_POSE[1], FOOT_RIGHT_POSE[2], 0, 0, 0))))

        # LEG LEFT
        HIP_LEFT_POSE = Pose_2_KUKA(kinect_model.Pose()*transl(-joints[PyKinectV2.JointType_HipLeft].Position.x*1000, -joints[PyKinectV2.JointType_HipLeft].Position.y*1000, joints[PyKinectV2.JointType_HipLeft].Position.z*1000))
        KNEE_LEFT_POSE = Pose_2_KUKA(kinect_model.Pose()*transl(-joints[PyKinectV2.JointType_KneeLeft].Position.x*1000, -joints[PyKinectV2.JointType_KneeLeft].Position.y*1000, joints[PyKinectV2.JointType_KneeLeft].Position.z*1000))
        ANKLE_LEFT_POSE = Pose_2_KUKA(kinect_model.Pose()*transl(-joints[PyKinectV2.JointType_AnkleLeft].Position.x*1000, -joints[PyKinectV2.JointType_AnkleLeft].Position.y*1000, joints[PyKinectV2.JointType_AnkleLeft].Position.z*1000))
        FOOT_LEFT_POSE = Pose_2_KUKA(kinect_model.Pose()*transl(-joints[PyKinectV2.JointType_FootLeft].Position.x*1000, -joints[PyKinectV2.JointType_FootLeft].Position.y*1000, joints[PyKinectV2.JointType_FootLeft].Position.z*1000))
        self.HIP_LEFT.setPoseAbs(KUKA_2_Pose(list((HIP_LEFT_POSE[0] + OFFSET_RGB, HIP_LEFT_POSE[1], HIP_LEFT_POSE[2], 0, 0, 0))))
        self.KNEE_LEFT.setPoseAbs(KUKA_2_Pose(list((KNEE_LEFT_POSE[0] + OFFSET_RGB, KNEE_LEFT_POSE[1], KNEE_LEFT_POSE[2], 0, 0, 0))))
        self.ANKLE_LEFT.setPoseAbs(KUKA_2_Pose(list((ANKLE_LEFT_POSE[0] + OFFSET_RGB, ANKLE_LEFT_POSE[1], ANKLE_LEFT_POSE[2], 0, 0, 0))))
        self.FOOT_LEFT.setPoseAbs(KUKA_2_Pose(list((FOOT_LEFT_POSE[0] + OFFSET_RGB, FOOT_LEFT_POSE[1], FOOT_LEFT_POSE[2], 0, 0, 0))))
        RDK.Render(True)


Operator = CloudSkeleton()
Operator.Circle()

--- Python program TestConnection ---
from robolink import *    # RoboDK API
from robodk import *      # Robot toolbox
RDK = Robolink()

robot = RDK.Item('KUKA')
tl = RDK.Item("Top Left")
bl = RDK.Item('Bottom Left')
# robot.setConnectionParams('169.254.98.120', 7000, '/', 'anonymous', '')
success = robot.Connect()
tar = tr(tl.Joints())
"""
    Change the position of the Joints because KUKA LWR IV+ has declared the third joint as an External Joint.
    KUKA LWR IV+ Joints = [A1, A2, E1, A3, A4, A5, A6] and RoboDK sends the joints as [A1, A2, A3, A4, A5, A6, E1]
"""
print(tr(bl.Joints()))
print(tr(tl.Joints()))
robot.MoveJ([tar[0, 0], tar[0, 1], tar[0, 3], tar[0, 4], tar[0, 5], tar[0, 6], tar[0, 2]])
tar = tr(bl.Joints())
robot.MoveJ([tar[0, 0], tar[0, 1], tar[0, 3], tar[0, 4], tar[0, 5], tar[0, 6], tar[0, 2]])
# robot.MoveJ(target)
robot.setSpeed(100)
RDK.Render(True)
# robot.MoveL()
# robot.MoveJ(home)
# robot.MoveJ([0, 90, 0, 0, 0, 0, 0])

--- Python program testRobotItem ---
from robolink import *    # RoboDK API
from robodk import *      # Robot toolbox
import time
RDK = Robolink()
RDK.Render(False)
t = time.time()
robot = None
for station in RDK.ItemList():
    for item in station.Childs():
        if item.type == ITEM_TYPE_ROBOT:
            robot = item
            break
    if robot is not None:
        break


print(time.time() - t)
RDK.Render(True)
robot.MoveJ([0, 90, 0, 0, 0, 0, 0])

--- Python program testJoints ---
from robolink import *    # RoboDK API
from robodk import *      # Robot toolbox
RDK = Robolink()

robot = RDK.Item("KUKA")
pose = RDK.Item("Top Left")
RDK.Render(True)
# Move Robot on Simulation Only
# RDK.setRunMode(1)  # Simulate only
# robot.MoveJ(pose)
# Move real robot
RDK.Render(False)
RDK.setRunMode(6)
tar = tr(pose.Joints())
print(Pose_2_KUKA(pose.Pose()))
"""
    Change the position of the Joints because KUKA LWR IV+ has declared the third joint as an External Joint.
    KUKA LWR IV+ Joints = [A1, A2, E1, A3, A4, A5, A6] and RoboDK sends the joints as [A1, A2, A3, A4, A5, A6, E1]
"""
robot.MoveJ([0, 90, 0, 0, 0, 0, 0])
# robot.MoveJ([tar[0, 0], tar[0, 1], tar[0, 3], tar[0, 4], tar[0, 5], tar[0, 6], tar[0, 2]])

--- Python program testRot ---
# Type help("robolink") or help("robodk") for more information
# Press F5 to run the script
# Documentation: https://robodk.com/doc/en/RoboDK-API.html
# Reference:     https://robodk.com/doc/en/PythonAPI/index.html
# Note: It is not required to keep a copy of this file, your python script is saved with the station
from robolink import *    # RoboDK API
from robodk import *      # Robot toolbox
RDK = Robolink()

br = RDK.Item("Bottom Right")
bl = RDK.Item("Bottom Left")
tl = RDK.Item("Top Left")
tr = RDK.Item("Top Right")

br_temp = Pose_2_KUKA(br.Pose())
bl_temp = Pose_2_KUKA(bl.Pose())
tl_temp = Pose_2_KUKA(tl.Pose())
tr_temp = Pose_2_KUKA(tr.Pose())
br.setPoseAbs(KUKA_2_Pose(list((br_temp[0], br_temp[1], br_temp[2], br_temp[3], br_temp[4], 45))))
bl.setPoseAbs(KUKA_2_Pose(list((bl_temp[0], bl_temp[1], bl_temp[2], bl_temp[3], bl_temp[4], bl_temp[5]))))
tl.setPoseAbs(KUKA_2_Pose(list((tl_temp[0], tl_temp[1], tl_temp[2], tl_temp[3], tl_temp[4], tl_temp[5]))))
tr.setPoseAbs(KUKA_2_Pose(list((tr_temp[0], tr_temp[1], tr_temp[2], tr_temp[3], tr_temp[4], tr_temp[5]))))

--- Python program testFabric ---
from robolink import *    # RoboDK API
from robodk import *      # Robot toolbox
RDK = Robolink()

br = RDK.Item('Bottom Right')
bl = RDK.Item('Bottom Left')
tl = RDK.Item('Top Left')
tr = RDK.Item('Top Right')
temp = br.Pose()
for i in [br, bl, tl, tr]:
    print((Pose_2_KUKA(i.PoseAbs())))

--- Python program quasi ---
from robolink import *    # RoboDK API
from robodk import *      # Robot toolbox
from numpy import pi as pi
import time
RDK = Robolink()
home = RDK.Item('Home')
hand = RDK.Item('Hand')
robot = RDK.Item('KUKA')
tl = RDK.Item('Top Left')
tar = RDK.Item('Target 8')
hand.setColor([255/255, 170/255, 127/255, 1])
hand.setPoseAbs(tl.PoseAbs()*roty(pi/2)*rotz(pi)*rotx(pi/2)*transl(-30, 0, 0))
robot.setSpeed(speed_linear=10*1000, speed_joints=110.0, accel_linear=-1, accel_joints=-1)
for i in range(7):
    hand.setPoseAbs(hand.PoseAbs()*rotx(pi/5))
    time.sleep(.4)
    hand.setPoseAbs(hand.PoseAbs()*rotx(-pi/5))
    time.sleep(.4)
    if i == 3:
        tar.setPoseAbs(KUKA_2_Pose(list((485, 250, 665, 45, 0, 180))))
        robot.MoveJ(tar)
        hand.setColor([1, 0, 0, 1])
        hand.setPoseAbs(hand.PoseAbs()*transl(15, 0, 0))
    if i == 6:
        robot.MoveJ(home)
        hand.setColor([255/255, 170/255, 127/255, 1])
        hand.setPoseAbs(hand.PoseAbs()*transl(-15, 0, 0))

--- Python program transient ---
from robolink import *    # RoboDK API
from robodk import *      # Robot toolbox
from numpy import pi as pi
import time

RDK = Robolink()
home = RDK.Item('Home')
hand = RDK.Item('Hand')
robot = RDK.Item('KUKA')
tl = RDK.Item('Top Left')
tar = RDK.Item('Target 8')
hand.setColor([255/255, 170/255, 127/255, 1])
robot.setSpeed(speed_linear=10*1000, speed_joints=110.0, accel_linear=-1, accel_joints=-1)
hand.setPoseAbs(tl.PoseAbs()*roty(pi/2)*rotz(pi)*rotx(pi/2)*transl(-400, 0, 0))
for i in range(6):
    hand.setPoseAbs(hand.PoseAbs()*transl(i*10, 0, 0))
    time.sleep(.5)
    if i == 3:
        tar.setPoseAbs(tl.PoseAbs()*transl(0, 0, -220))
        robot.MoveJ(tar)
        hand.setColor([1, 0, 0, 1])
        for j in range(5):
            hand.setPoseAbs(hand.PoseAbs()*transl(15, 0, 0))
            tar.setPoseAbs(tar.PoseAbs()*transl(0, 0, 15))
            robot.MoveJ(tar)
        hand.setPoseAbs(hand.PoseAbs()*transl(25, 0, 0))
        hand.setPoseAbs(hand.PoseAbs()*transl(25, 0, 0))
        hand.setPoseAbs(hand.PoseAbs()*transl(20, 0, 0))
        hand.setColor([255/255, 170/255, 127/255, 1])
        robot.MoveJ(home)
        hand.setColor([255/255, 170/255, 127/255, 1])

--- Python program testJointLimits ---
from robolink import *    # RoboDK API
from robodk import *      # Robot toolbox
RDK = Robolink()

robot = RDK.Item('KUKA')

robot.MoveJ([175, 25, 40, 50, 60, 70, 80])
